FUNCTION_BLOCK UINT_DEMUX_N (* Basic Function Block Type *)
  (* Standard: 61499-2 *)
  (* Version 0.0, 2015-11-03, 4DIAC-IDE, 4DIAC-Consortium *)
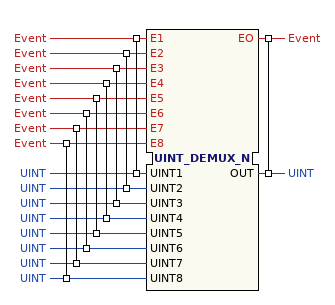
  EVENT_INPUT
    E1 WITH UINT1;
    E2 WITH UINT2;
    E3 WITH UINT3;
    E4 WITH UINT4;
    E5 WITH UINT5;
    E6 WITH UINT6;
    E7 WITH UINT7;
    E8 WITH UINT8;
  END_EVENT
  EVENT_OUTPUT
    EO WITH OUT;
  END_EVENT
  VAR_INPUT
    UINT1 : UINT;
    UINT2 : UINT;
    UINT3 : UINT;
    UINT4 : UINT;
    UINT5 : UINT;
    UINT6 : UINT;
    UINT7 : UINT;
    UINT8 : UINT;
  END_VAR
  VAR_OUTPUT
    OUT : UINT;
  END_VAR
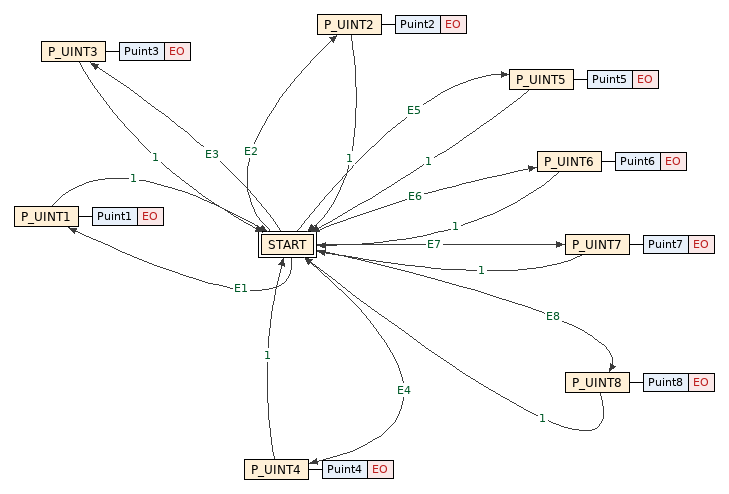
  EC_STATES
    START; (* Initial State *)
    P_UINT3 : Puint3 -> EO; (* Initialization *)
    P_UINT1 : Puint1 -> EO; (* Normal execution *)
    P_UINT2 : Puint2 -> EO;
    P_UINT4 : Puint4 -> EO;
    P_UINT5 : Puint5 -> EO;
    P_UINT6 : Puint6 -> EO;
    P_UINT7 : Puint7 -> EO;
    P_UINT8 : Puint8 -> EO;
  END_STATES
  EC_TRANSITIONS
    START TO P_UINT3 := E3;
    P_UINT3 TO START := 1;
    START TO P_UINT1 := E1;
    P_UINT1 TO START := 1;
    P_UINT2 TO START := 1;
    START TO P_UINT2 := E2;
    P_UINT4 TO START := 1;
    START TO P_UINT4 := E4;
    START TO P_UINT5 := E5;
    P_UINT5 TO START := 1;
    START TO P_UINT6 := E6;
    P_UINT6 TO START := 1;
    START TO P_UINT7 := E7;
    P_UINT7 TO START := 1;
    START TO P_UINT8 := E8;
    P_UINT8 TO START := 1;
  END_TRANSITIONS
  ALGORITHM Puint1 IN ST: (* Print UINT1 -> OUT *)
OUT:=UINT1;
  END_ALGORITHM
  ALGORITHM Puint2 IN ST: (* Print UINT2 -> OUT *)
OUT:=UINT2;
  END_ALGORITHM
  ALGORITHM Puint3 IN ST: (* Print UINT3 -> OUT *)
OUT:=UINT3;
  END_ALGORITHM
  ALGORITHM Puint4 IN ST: (* Print UINT4 -> OUT *)
OUT:=UINT4;
  END_ALGORITHM
  ALGORITHM Puint5 IN ST: (* Print UINT5 -> OUT *)
OUT:=UINT5;
  END_ALGORITHM
  ALGORITHM Puint6 IN ST: (* Print UINT6 -> OUT *)
OUT:=UINT6;
  END_ALGORITHM
  ALGORITHM Puint7 IN ST: (* Print UINT7 -> OUT *)
OUT:=UINT7;
  END_ALGORITHM
  ALGORITHM Puint8 IN ST: (* new algorithm *)
OUT:=UINT8;
  END_ALGORITHM
END_FUNCTION_BLOCK
